RESOURCE RES0 : EMB_RES_ECO
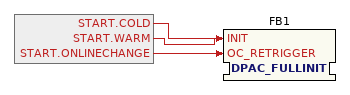
  (* NVPP_Application *)
  FBS
    FB1 : DPAC_FULLINIT;
  END_FBS
  EVENT_CONNECTIONS
    START.COLD TO FB1.INIT;
    START.WARM TO FB1.INIT;
    START.ONLINECHANGE TO FB1.OC_RETRIGGER;
  END_CONNECTIONS
END_RESOURCE
